// TIA Portal V20 export
FUNCTION_BLOCK "FB_LaserOperation"   // FB431, SCL
{ S7_Optimized_Access := 'TRUE' }
// stored: AutoNumber false, MemoryReserve 100, SetENOAutomatically false
   VAR
      sLaserTimeCh1 : "FB_TimeCounter";
      sLaserCycleTimeCh1 { S7_SetPoint := 'True'} : Int;
   END_VAR
BEGIN
   REGION Description header 
       //==================================================================================
       // POSALUX Swiss SA / (C) Copyright 2024
       //----------------------------------------------------------------------------------
       // Title: Laser AirProcess
       // Comment/Function: 
       //
       // Author: Gowsigan SRITHARAN
       // Engineering: TIA Portal v17
       //----------------------------------------------------------------------------------
       // Change log table:
       // Version  | Date     | Expert in charge | Changes applied
       // ---------|----------|------------------|------------------------------------
       // 00.00.01 | 20241205 | GSR              | First released version
       // ==================================================================================
   END_REGION

   REGION Head Laser Circuit breaker
       IF NOT "DB_DigitalInputs".sHeadLaserBreaker.sSWStatus THEN
           "LBP_AlarmMsgs".UserA[0].A70UUxx[2] := TRUE;
       END_IF;
   END_REGION

   REGION Head_Laser start and stop
       "DB_DigitalOutputs".sHeadLaserStart.sSWStatus := "DB_PowerOn".sMachineReadySoft;
       "DB_DigitalOutputs".sHeadLaserStop.sSWStatus  := "DB_PowerOn".sMachineReadySoft;
   END_REGION

   REGION LED laser button 
       IF ("DB_DataFromSafety".ShutterOpened
           AND NOT "DB_DataFromSafety".ShutterClosed)
           OR "DB_McpKeyboardSignals".sLightTest.sKeySWStatus THEN  // Test Lamp
           "DB_McpKeyboardSignals".sRemoteOpenShutter.sLedSWStatus := TRUE;
       ELSIF "DB_DataFromSafety".ShutterClosed AND NOT "DB_DataFromSafety".ShutterOpened THEN
           IF "DB_DataFromSafety".ShutterReadyToOpen THEN
               // Ready to open -> slow blinking
               "DB_McpKeyboardSignals".sRemoteOpenShutter.sLedSWStatus := "Clock_0.5Hz";
           ELSIF "DB_DataFromSafety".OpenShutter THEN
               // Ready to open -> quick blinking
               "DB_McpKeyboardSignals".sRemoteOpenShutter.sLedSWStatus := "Clock_2Hz";
           ELSE
               // Close -> off
               "DB_McpKeyboardSignals".sRemoteOpenShutter.sLedSWStatus := FALSE;
           END_IF;
       ELSE
           // Close -> off
           "DB_McpKeyboardSignals".sRemoteOpenShutter.sLedSWStatus := FALSE;
       END_IF;
   END_REGION

   REGION Laser Key ON / Shutter closed
       "DB_HMIStatus".KeyLaserOn := "DB_DataFromSafety".iKeyLaserOn;
       "DB_HMIStatus".Shutter_laser_closed := "DB_DigitalInputs".sShutterClosed.sSWStatus OR NOT "DB_DataFromSafety".iKeyLaserOn;
   END_REGION


   REGION Laser Cycle Time
       #sLaserTimeCh1(iStart := "LBP_Chan1".MDyn[71],                        // M71 : Start calculation laser time 
                      iReset := "LBP_Chan1".MDyn[68] OR "MCP1_In".reset);    // M68 : Reset calculation laser time 
       #sLaserCycleTimeCh1 := #sLaserTimeCh1.ioMinutesCumul;
   END_REGION
END_FUNCTION_BLOCK
